TYPE MppcConfigs :
STRUCT
	C13336MppcConfigWide   : C13336MppcConfig;
	C13336MppcConfigNarrow : C13336MppcConfig;
END_STRUCT
END_TYPE

(* stored: Version 1.1.0.1, ProductVersion 3.1.4024.3
   DUT MppcConfigs: Id {63b7a9e7-8a1c-4e12-a93a-576f7a753afb} *)
